// TIA Portal V17 export
// export: Created 2025-06-26T06:49:25.5830311Z, ExportSetting WithDefaults, DisplayName Totally Integrated Automation Portal, DisplayVersion V17 Update 8, DisplayName TIA Portal Openness, DisplayVersion V17 Update 8, DisplayName TIA Portal Version Control Interface, DisplayVersion V17, DisplayName STEP 7 Professional, DisplayVersion V17 Update 8, DisplayName STEP 7 Safety, DisplayVersion V17 Update 6, DisplayName WinCC Advanced, DisplayVersion V17 Update 8
DATA_BLOCK "DB_Regulators"   // DB18
{ S7_Optimized_Access := 'FALSE' }
AUTHOR : Heaten
VERSION : 0.1
// stored: AutoNumber true, DBAccessibleFromOPCUA true, DBAccessibleFromWebserver true, IsOnlyStoredInLoadMemory false, IsWriteProtectedInAS false
   VAR RETAIN
      CabinetTemperature : "stTemperatureController2";   // Regulates PLC cabinet temperature
      OilHeating { S7_SetPoint := 'True'} : "stOilHeater";   // Regulates compressor oil sump temperature
      ContainerVentilation { S7_SetPoint := 'True'} : "stPI_Regulator";   // Regulates container air temperature
      CPCPressure { S7_SetPoint := 'True'} : "stPI_Regulator";   // Regulates CPC pressure
      CPCReservoir { S7_SetPoint := 'True'} : "stOnOffRegulator";   // Regulates CPC reservoir level
      CPCReservoirPlanB { S7_SetPoint := 'True'} : "stProgressivePeriodicRegulator4";   // Regulates CPC reservoir level (Plan B)
      ShaftSealCirculation { S7_SetPoint := 'True'} : "stCirculationPump";   // Barrier fluid circulation
      ShaftSealCooler { S7_SetPoint := 'True'} : "stOnOffRegulator";   // Barrier fluid temperature
      ShaftSealRecharge { S7_SetPoint := 'True'} : "stOnOffRegulator";   // Barrier fluid pressure
      OilSeparator { S7_SetPoint := 'True'} : "stOilSeparator";   // Regulates oil level in oil separator
      LubricationPriming { S7_SetPoint := 'True'} : "stPrimerPump";   // Compressor lubrication priming
      PerformanceControl { S7_SetPoint := 'True'} : "stPerformanceControl";   // Compressor speed control
      SuperheatControl { S7_SetPoint := 'True'} : "stSuperheatControl";   // Regulates superheat
      PinchControl { S7_SetPoint := 'True'} : "stPinchControl";   // Regulates pinch
      PurgeControl { S7_SetPoint := 'True'} : "stPurgeControl";   // Handles purging of compressor suction manifold
      FilterDryer { S7_SetPoint := 'True'} : "stFilterDryer";   // Runs filter dryer circuit
      OilRecovery { S7_SetPoint := 'True'} : "stOilRecovery";   // Runs oil recovery circuit
      RecuperatorBypass { S7_SetPoint := 'True'} : "stNullRegulator";   // Runs recuperator bypass
      HeatSourceCycle { S7_SetPoint := 'True'} : "stTrackingRegulator";
      HeatSourceCyclePIP { S7_SetPoint := 'True'} : "stPIP_Regulator";   // Regulates heat exchanger temperature rise
      DischargeAccumulator { S7_SetPoint := 'True'} : "stOnOffRegulator3";   // Discharge accumulator return
      SuctionAccumulator { S7_SetPoint := 'True'} : "stOnOffRegulator3";   // Suction accumulator return
      HeatboosterSetpoint { S7_SetPoint := 'True'} : Real;   // TEST: selected setpoint
      RegulationTarget : Int;   // TEST: selected regulation target
   END_VAR
BEGIN
   CabinetTemperature.bEnable := true;
   CabinetTemperature.fHeatingSetpoint := 15.0;
   CabinetTemperature.fCoolingSetpoint := 40.0;
   OilHeating.fOilSuperheat := 15.0;
   OilHeating.Controller.bEnable := true;
   OilHeating.Controller.fHysteresis := 2.0;
   ContainerVentilation.bEnable := false;
   CPCPressure.bEnable := false;
   CPCReservoir.bEnable := true;
   CPCReservoir.fSetpoint := 60.0;
   CPCReservoirPlanB.tManualPeriod := T#10m;
   CPCReservoirPlanB.tOnTime := T#15s;
   CPCReservoirPlanB.Param.Limit[0] := 400.0;
   CPCReservoirPlanB.Param.Limit[1] := 500.0;
   CPCReservoirPlanB.Param.Limit[2] := 600.0;
   CPCReservoirPlanB.Param.Limit[3] := 700.0;
   CPCReservoirPlanB.Param.Period[0] := T#20m;
   CPCReservoirPlanB.Param.Period[1] := T#14m;
   CPCReservoirPlanB.Param.Period[2] := T#7m;
   CPCReservoirPlanB.Param.Period[3] := T#1m;
   ShaftSealCirculation.bEnable := true;
   ShaftSealCooler.bEnable := true;
   ShaftSealCooler.fSetpoint := 97.5;
   ShaftSealCooler.fHysteresis := 5.0;
   ShaftSealRecharge.bEnable := true;
   ShaftSealRecharge.fSetpoint := 1120.0;
   ShaftSealRecharge.fHysteresis := 200.0;
   // OilSeparator.Stage1 : Level control Stage 1
   // OilSeparator.Stage2 : Level control Stage 2
   LubricationPriming.fMotorSpeed := 2830.0;
   LubricationPriming.fMotorTorqueLimit := 70.0;
   LubricationPriming.Controller.bEnable := true;
   LubricationPriming.Controller.fSetpoint := 140.0;
   LubricationPriming.Controller.fHysteresis := 80.0;
   PerformanceControl.Settings.HeatSink.Control_Active := true;
   PerformanceControl.Settings.HeatSink.Kp := 16.0;
   PerformanceControl.Settings.HeatSource.Control_Active := false;
   PerformanceControl.Settings.HeatSource.Kp := -4.0;
   PerformanceControl.Settings.VariableControl.Control_Active := false;
   PerformanceControl.Settings.Config.MinimumPerformanceRequirement := 30.0;
   PerformanceControl.Settings.Config.MaximumAdditionalSuperheat := 35.0;
   PerformanceControl.Settings.Config.INCREASEWITHNORESTRICTION := 0.2;
   SuperheatControl.bEnable := true;
   SuperheatControl.Regulator.fFeedbackHysteresis := 15.0;
   SuperheatControl.Regulator.fOutMax := 100.0;
   SuperheatControl.Regulator.fOutMin := -50.0;
   SuperheatControl.Regulator.Kp := 0.8;
   SuperheatControl.Regulator.Tn := 35.0;
   SuperheatControl.Regulator.Tv := 0.0;
   SuperheatControl.Regulator.T1 := 0.0;
   SuperheatControl.fineTuningRecTarget := 0.65;
   SuperheatControl.ExponentialPinchFactor := 21.6;
   PinchControl.bEnable := true;
   PinchControl.Regulator.fOutMax := 100.0;
   PinchControl.Regulator.Kp := 1.0;
   PinchControl.Regulator.Tn := 4.0;
   PinchControl.Regulator.Tv := 16.0;
   PinchControl.Regulator.T1 := 0.0;
   PurgeControl.nPurgeCycles := 3;
   PurgeControl.bEnable := true;
   PurgeControl.Purge.nPurgeType := 0;
   PurgeControl.Purge.tPurgeTime := T#15s;
   PurgeControl.Purge.fPurgeDeltaP := 35.0;
   PurgeControl.Spin.tSpinTime := T#20s;
   PurgeControl.Spin.fSpinSpeed := 250.0;
   PurgeControl.Spin.fSpinRamp := 50.0;
   FilterDryer.fFixedOutput := 50.0;
   FilterDryer.Controller.tOnTime := T#3m;
   FilterDryer.Controller.tPeriod := T#30m;
   OilRecovery.nRunRatio := 5;
   OilRecovery.Controller.tOnTime := T#1m;
   OilRecovery.Controller.tStartDelay := T#5s;
   // HeatSourceCyclePIP.fPV : [C] Heat source temperature
   // HeatSourceCyclePIP.fPVvel : [K/sec] Heat source temperature rate of change
   HeatSourceCyclePIP.fSP := 120.0;   // [C] Heat source temperature setpoint
   HeatSourceCyclePIP.fOutMax := 100.0;   // [%] Max valve position
   HeatSourceCyclePIP.fOutMin := 0.0;   // [%] Min valve position
   HeatSourceCyclePIP.fVelMax := 5.0;   // [K/min] Max positive temperature rate of change
   HeatSourceCyclePIP.fVelMin := -5.0;   // [K/min] Max negative temperature rate of change
   // HeatSourceCyclePIP.fOut : [%] Valve position
   // HeatSourceCyclePIP.fManualValue : [%] Manual manipulated value
   HeatSourceCyclePIP.Kp := 1.0;   // Proportional gain temperature (C/s per C)
   HeatSourceCyclePIP.Tn := 0.0;   // Integral gain temperature
   HeatSourceCyclePIP.KpVel := 15.0;   // Proportional gain temperature rate of change (% per C/s)
   HeatSourceCyclePIP.TnVel := 75.0;
   HeatSourceCyclePIP.fFeedbackHysteresis := 0.2;
END_DATA_BLOCK
